// SIMATIC STEP 7 (V5.x) project StarDeltaMotor
// CPU: CPU 314C-2 DP
// station: Hardware
// station: SIMATIC 300(1)
// station: P_ADR_BUS
// program: S7 Program(1)

SYMBOL_TABLE
"Stop"	I 0.1	BOOL
"Main Start"	Q 0.0	BOOL
"Star"	Q 0.1	BOOL
"Delat"	Q 0.2	BOOL
END_SYMBOL_TABLE

ORGANIZATION_BLOCK OB 1
TITLE = "Starting a Motor first with Star and then Delta"
VERSION : 0.1
VAR_TEMP
  OB1_EV_CLASS : BYTE ;	//Bits 0-3 = 1 (Coming event), Bits 4-7 = 1 (Event class 1)
  OB1_SCAN_1 : BYTE ;	//1 (Cold restart scan 1 of OB 1), 3 (Scan 2-n of OB 1)
  OB1_PRIORITY : BYTE ;	//Priority of OB Execution
  OB1_OB_NUMBR : BYTE ;	//1 (Organization block 1, OB1)
  OB1_RESERVED_1 : BYTE ;	//Reserved for system
  OB1_RESERVED_2 : BYTE ;	//Reserved for system
  OB1_PREV_CYCLE : INT ;	//Cycle time of previous OB1 scan (milliseconds)
  OB1_MIN_CYCLE : INT ;	//Minimum cycle time of OB1 (milliseconds)
  OB1_MAX_CYCLE : INT ;	//Maximum cycle time of OB1 (milliseconds)
  OB1_DATE_TIME : DATE_AND_TIME ;	//Date and time OB1 started
END_VAR
BEGIN
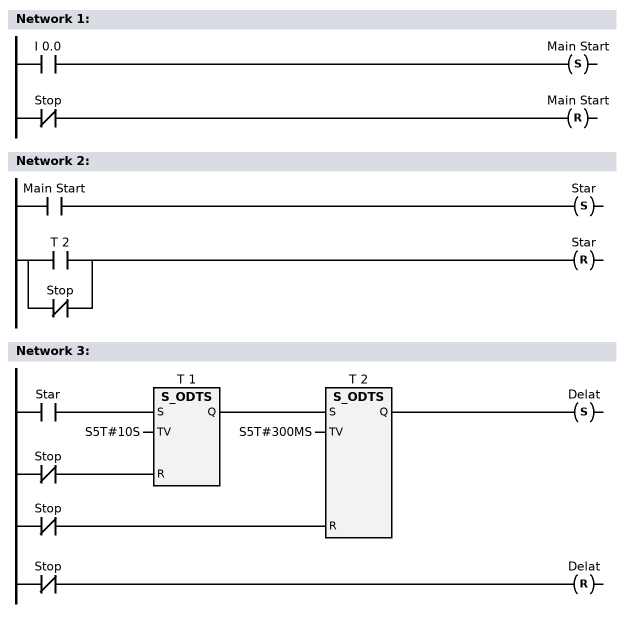
NETWORK
TITLE =
      A     I 0.0;
      S     "Main Start";
      AN    "Stop";
      R     "Main Start";
      NOP   0;
NETWORK
TITLE =
      A     "Main Start";
      S     "Star";
      A(;
      O     T 2;
      ON    "Stop";
      );
      R     "Star";
      NOP   0;
NETWORK
TITLE =
      A(;
      A(;
      A     "Star";
      L     S5T#10S;
      SS    T 1;
      AN    "Stop";
      R     T 1;
      NOP   0;
      NOP   0;
      A     T 1;
      );
      L     S5T#300MS;
      SS    T 2;
      AN    "Stop";
      R     T 2;
      NOP   0;
      NOP   0;
      A     T 2;
      );
      S     "Delat";
      AN    "Stop";
      R     "Delat";
      NOP   0;
END_ORGANIZATION_BLOCK
